FUNCTION_BLOCK FB_DIV_DINT (* DINT Division *)
  (* Standard: 61499-1-D.1; Classification: Math *)
  (* Version 0.1, 2001-08-05, JHC, Rockwell Automation, XML version; subclassed from FBFunctionQS2. *)
  (* Version 0.0, 1997-09-11, JHC, Rockwell Automation, Original (SRC) version. *)
  (* Compiler header: package fb.rt.math; *)
  (* Compiler classdef: class FB_DIV_DINT extends FBFunctionQS2 *)
  (* Compiler Java IBM VisualAge 3.0 *)
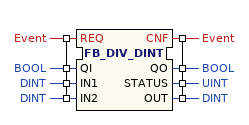
  EVENT_INPUT
    REQ WITH QI, IN1, IN2;
  END_EVENT
  EVENT_OUTPUT
    CNF WITH QO, STATUS, OUT;
  END_EVENT
  VAR_INPUT
    QI : BOOL; (* Event Qualifier *)
    IN1 : DINT; (* Dividend *)
    IN2 : DINT; (* Divisor *)
  END_VAR
  VAR_OUTPUT
    QO : BOOL; (* Output Qualifier *)
    STATUS : UINT; (* Operation Status *)
    OUT : DINT; (* Quotient *)
  END_VAR
END_FUNCTION_BLOCK
